% RSLogix 500 project Temperature Control System.RSS, saved by version 8.30.00.16 %
PROJECT "UNTITLED"    % processor: Bul.1763 MicroLogix 1100 Series B %

PROGRAM FILES
  LAD 2   3 rungs

DATA FILES
  O0 OUTPUT  4 elements
  I1 INPUT  6 elements
  S2 STATUS  66 elements
  B3 BINARY  1 elements
  T4 TIMER  1 elements
  C5 COUNTER  1 elements
  R6 CONTROL  1 elements
  N7 INTEGER  1 elements
  F8 FLOAT  1 elements

LADDER 2
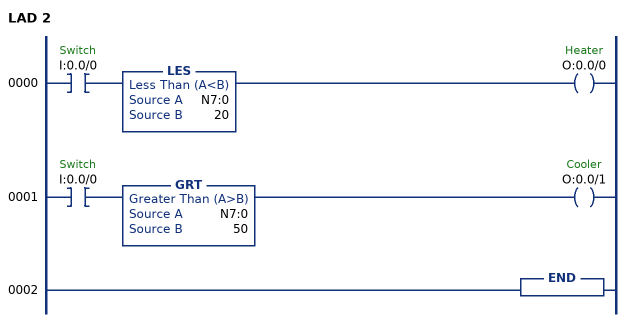
% Rung: 0 %
SOR XIC I:0.0/0 LES N7:0 20 OTE O:0.0/0 EOR
%   I:0.0/0  "Switch" %
%   O:0.0/0  "Heater" %
% Rung: 1 %
SOR XIC I:0.0/0 GRT N7:0 50 OTE O:0.0/1 EOR
%   I:0.0/0  "Switch" %
%   O:0.0/1  "Cooler" %
% Rung: 2 %
SOR END EOR

DATA TABLE (non-zero values as saved)
DATA N7
% N7:0 % 51
